{attribute 'qualified_only'}
{attribute 'strict'}
{attribute 'conditionalshow'}
{attribute 'to_string'}
TYPE E_Scope :
(
	eLog			:= 0,
	eLogger			:= 1,
	eScoped			:= 2,
	eTask			:= 3
) BYTE;
END_TYPE

(* stored: Version 1.1.0.1, ProductVersion 3.1.4024.6
   DUT E_Scope: Id {0cb1f182-209d-44d8-b9c4-d492da6de2ee} *)
